// TIA Portal V20 export
DATA_BLOCK "DB_McpKeyboardSignals"   // DB421
// stored: AutoNumber false, InstanceOfName FB_McpKeyboardSignals, InstanceOfType FB
"FB_McpKeyboardSignals"
   // VAR
   //    sK1_Powermeter : "FB_McpKeysSignals";
   //    sK2_GasAssist : "FB_McpKeysSignals";
   //    sK3_KeySaveParam : "FB_McpKeysSignals";
   //    sK4_GripperUndrilledPart : "FB_McpKeysSignals";
   //    sK5_GripperDrilledPart : "FB_McpKeysSignals";
   //    sK6_SITestStop : "FB_McpKeysSignals";
   //    sK7_FixtureClamp : "FB_McpKeysSignals";
   //    sK8_FixtureVacuum : "FB_McpKeysSignals";
   //    sK9_Aspiration : "FB_McpKeysSignals";
   //    sK10_LoaderAuto : "FB_McpKeysSignals";
   //    sK11_LoaderSemiAuto : "FB_McpKeysSignals";
   //    sK12_ObservationCamera : "FB_McpKeysSignals";
   //    sK13_MainDoor : "FB_McpKeysSignals";
   //    sK14_WarmUp : "FB_McpKeysSignals";
   //    sK15_MachineLight : "FB_McpKeysSignals";
   //    sStartCycle { S7_SetPoint := 'True'} : "FB_McpKeysSignals";
   //    sAlarmReset { S7_SetPoint := 'True'} : "FB_McpKeysSignals";
   //    sPowerOFF { S7_SetPoint := 'True'} : "FB_McpKeysSignals";
   //    sShutdownPC { S7_SetPoint := 'True'} : "FB_McpKeysSignals";
   //    sLightTest { S7_SetPoint := 'True'} : "FB_McpKeysSignals";
   //    sPowerON { S7_SetPoint := 'True'} : "FB_McpKeysSignals";
   //    sRemoteOpenShutter { S7_SetPoint := 'True'} : "FB_McpKeysSignals";
   //    sAx10_LaserArea { S7_SetPoint := 'True'} : "FB_McpKeysSignals";
   //    sAx11_ChannelSelection { S7_SetPoint := 'True'} : "FB_McpKeysSignals";
   // END_VAR
BEGIN
END_DATA_BLOCK
